Yaskawa INFORM job: R1_W17,20,22(0,0)OK-KM.JBI

/JOB
//NAME R1_W17,20,22(0,0)OK-KM
///FOLDERNAME KRIS-SCIANA
//POS
///NPOS 121,121,0,7,0,0
///TOOL 0
///POSTYPE PULSE
///PULSE
C00000=-189615,-139320,-99333,22908,80634,5417
C00001=-195814,-97363,-54861,18109,45254,4013
C00002=-195342,-89844,-49219,17779,45528,4291
C00003=-194630,-83582,-43444,17553,45059,4532
C00004=-193782,-82947,-43197,17110,45053,4932
C00005=-194630,-83582,-43444,17553,45059,4532
C00006=-194630,-82704,-41910,17701,44589,4439
C00007=-199143,-72536,-44097,19526,61527,3376
C00008=-199513,-75125,-46608,19573,61817,3281
C00009=-200501,-81674,-52788,19719,62464,3007
C00010=-207304,-71791,-24407,35263,30060,5319
C00011=-207149,-64591,-18647,35001,30129,5478
C00012=-204869,-60384,-14661,33643,29035,6515
C00013=-203452,-59589,-14281,32383,28672,7366
C00014=-204869,-60384,-14661,33643,29035,6515
C00015=-204869,-59185,-12583,34316,28482,6172
C00016=-204869,-60384,-14661,33643,29035,6515
C00017=-215068,-50959,-15594,37598,47140,3454
C00018=-215285,-50166,-15160,37584,47344,3432
C00019=-214356,-52683,-17577,37193,47111,3828
C00020=-214795,-55416,-20188,37217,47456,3749
C00021=-215972,-62244,-26544,37355,48272,3487
C00022=-217673,2073,-2688,-67811,68721,47040
C00023=-218977,3637,818,-67445,65858,48607
C00024=-219089,4523,1579,-67431,65778,48594
C00025=-218977,3637,818,-67445,65858,48607
C00026=-216731,7597,16575,-81534,66129,55483
C00027=-216731,8242,18363,-81863,65994,55863
C00028=-217587,5856,11870,-80689,65886,54435
C00029=-224554,-2275,-18337,-52519,68642,41010
C00030=-225245,-2625,-18625,-52307,68252,40859
C00031=-224554,-2275,-18337,-52519,68642,41010
C00032=-223707,-4148,-20438,-52681,69325,41069
C00033=-222614,-33118,-39506,-62827,46949,50873
C00034=-225738,-29129,-36820,-61092,45172,49948
C00035=-227041,-26413,-34946,-60254,44485,49501
C00036=-227207,-24592,-33670,-60039,44458,49378
C00037=-226942,-27472,-35680,-60383,44499,49577
C00038=-228936,-27670,-24586,-81470,38078,57242
C00039=-229553,-27860,-24718,-81378,37631,57193
C00040=-228393,-29098,-27492,-80247,38667,56535
C00041=-227197,-30656,-28257,-80893,39459,56892
C00042=-224091,-34376,-30000,-82400,41545,57754
C00043=-172648,-102914,-69268,-89134,45979,57650
C00044=-78280,-132294,-70134,-65050,82728,51954
C00045=231366,-50529,-85532,-14348,118547,17853
C00046=231331,-51716,-35505,-12276,87907,21200
C00047=229315,-48570,-29966,-12403,85849,20709
C00048=227923,-45606,-26730,-12487,85179,20296
C00049=227923,-45208,-25708,-12491,84764,20337
C00050=228522,-47247,-27691,-12456,85024,20518
C00051=199703,-85274,-38967,20911,45379,18978
C00052=198515,-84591,-38717,21283,45850,18535
C00053=199928,-86071,-39510,20852,45254,19054
C00054=200123,-88829,-42015,20735,45324,19162
C00055=200648,-95812,-48167,20467,45386,19423
C00056=223036,-16803,-12767,15055,51086,10558
C00057=223001,-10097,-5312,15317,49989,10370
C00058=221760,-6374,-575,16251,49262,9685
C00059=221760,-6023,569,16378,48758,9599
C00060=222987,-7382,-2234,15435,49509,10287
C00061=229840,2245,989,-2824,59416,19535
C00062=229297,2441,1158,-2588,59396,19324
C00063=229875,1901,-451,-2819,60125,19531
C00064=227161,1886,-1137,2630,57624,16683
C00065=227281,3372,123,2575,57604,16729
C00066=227129,1132,-3217,2621,58516,16692
C00067=227372,-1279,-6275,2488,59150,16802
C00068=228006,-7193,-13686,2154,60653,17078
C00069=231366,-50529,-85532,-14348,118547,17853
C00070=-77958,-132702,-65854,-64701,82399,51968
C00071=-138956,-107357,-30738,-74002,40113,39794
C00072=-140081,-59966,15635,-79359,38411,42592
C00073=-208206,-45897,20537,87676,15751,-45063
C00074=-207960,-49182,17085,86162,15646,-44311
C00075=-111965,-46340,36967,-74147,51082,48825
C00076=-82556,-17668,73730,-64807,60582,55576
C00077=-75120,-43857,42150,-58556,66417,53756
C00078=-148664,-83770,1112,-87446,33384,44594
C00079=-176147,-61139,7237,-80789,19096,34535
C00080=-180433,-47939,16447,-77543,16865,32116
C00081=-208028,-46200,20021,87142,15660,-44778
C00082=-207778,-49477,16583,85630,15556,-44027
C00083=-140712,-22447,70317,-98622,37333,53286
C00084=-126468,-40765,51508,-87063,43300,51710
C00085=-78280,-117024,-65873,-65050,51337,51954
C00086=204216,-84591,-49290,-51682,73827,23894
C00087=234941,-57799,-26790,-47858,90257,30629
C00088=199972,-101228,-53558,-4187,23841,10008
C00089=189033,-76626,-31890,10620,23559,1426
C00090=189033,-76626,-31890,10620,23559,1426
C00091=188864,-64798,-20049,11393,22392,1030
C00092=229125,-13360,-10863,-46798,76248,11937
C00093=228748,-14451,-12356,-46697,76301,11724
C00094=158433,-60990,9751,67845,21798,-31218
C00095=158927,-83907,-11161,65252,21999,-29865
C00096=192853,-97920,-56876,4665,27613,4814
C00097=204487,-80585,-57206,-6895,36944,11799
C00098=205889,-64287,-49388,-7540,40605,12218
C00099=203918,-48473,-33642,-6113,38883,11330
C00100=229115,-13382,-10880,-46798,76242,11935
C00101=228739,-14472,-12373,-46696,76295,11722
C00102=188637,-64887,-20002,11738,22348,831
C00103=195288,-76653,-33683,2057,24178,6381
C00104=224712,-65391,-70566,-27443,33176,35029
C00105=213770,-36542,-34460,77474,7084,-9175
C00106=213911,-28559,-27626,78111,6960,-9462
C00107=226738,-22872,-44138,-26151,38823,34122
C00108=225474,-24610,-45368,-24938,38325,33575
C00109=213819,-17629,4736,154767,14347,-43948
C00110=214272,-23134,1814,157793,15117,-45305
C00111=214272,-33613,-26176,108147,6753,-22913
C00112=214465,-33157,-25875,108062,6602,-22875
C00113=214484,-33168,-25884,108106,6590,-22894
C00114=214462,-14862,18245,165247,20516,-48770
C00115=217554,-35080,-3939,169426,16769,-50400
C00116=215729,-48765,-65733,21008,15669,16203
C00117=214456,-35235,-57699,21691,17865,16014
C00118=214365,-32785,-25079,110368,6760,-23908
C00119=218232,-57197,-39676,150711,6696,-41886
C00120=106022,-135537,-66235,115408,55550,-32403
BC00000=365100,2604,568777
BC00001=396813,15,501820
BC00002=396813,15,501820
BC00003=396813,15,501820
BC00004=396813,15,501820
BC00005=396813,15,501820
BC00006=396813,15,501820
BC00007=396813,15,501820
BC00008=396813,15,501820
BC00009=396813,15,501820
BC00010=289343,15,994506
BC00011=289343,15,994506
BC00012=289344,16,994504
BC00013=289344,16,994504
BC00014=289344,16,994504
BC00015=289344,16,994504
BC00016=289344,16,994504
BC00017=289343,15,994506
BC00018=289343,15,994506
BC00019=289343,15,994506
BC00020=289343,15,994506
BC00021=289343,15,994506
BC00022=398117,15,691553
BC00023=398117,15,691553
BC00024=398117,15,691553
BC00025=398117,15,691553
BC00026=398117,15,691553
BC00027=398117,15,691553
BC00028=398117,15,691553
BC00029=398117,15,691553
BC00030=398117,15,691553
BC00031=398117,15,691553
BC00032=398117,15,691553
BC00033=398174,15,1075175
BC00034=398174,15,1075175
BC00035=398174,15,1075175
BC00036=398174,15,1075175
BC00037=398174,15,1075175
BC00038=398174,15,1075175
BC00039=398174,15,1075175
BC00040=398174,15,1075175
BC00041=398174,15,1075175
BC00042=398174,15,1075175
BC00043=398174,15,1075175
BC00044=398174,15,1075175
BC00045=398174,29742,582568
BC00046=398174,29742,582568
BC00047=398174,29742,582568
BC00048=398174,29742,582568
BC00049=398174,29742,582568
BC00050=398174,29742,582568
BC00051=398174,29742,582568
BC00052=398174,29742,582568
BC00053=398174,29742,582568
BC00054=398174,29742,582568
BC00055=398174,29742,582568
BC00056=398174,24813,868263
BC00057=398174,24813,868263
BC00058=398174,24813,868263
BC00059=398174,24813,868263
BC00060=398174,24813,868263
BC00061=398174,24813,868263
BC00062=398174,24813,868263
BC00063=398174,24813,868263
BC00064=398174,24813,868263
BC00065=398174,24813,868263
BC00066=398174,24813,868263
BC00067=398174,24813,868263
BC00068=398174,24813,868263
BC00069=398174,29742,582568
BC00070=398174,15,1075175
BC00071=282653,15,945445
BC00072=282653,15,945445
BC00073=320510,15,961588
BC00074=320510,15,961588
BC00075=282653,15,931025
BC00076=282653,15,914571
BC00077=282653,15,945445
BC00078=282653,15,1075175
BC00079=282653,15,1075175
BC00080=282654,15,1075174
BC00081=282653,15,1075175
BC00082=282653,15,1075175
BC00083=282653,15,1075175
BC00084=282653,15,1075175
BC00085=398174,15,1075175
BC00086=344180,85519,956119
BC00087=344180,85519,956119
BC00088=331941,89333,813920
BC00089=331941,89333,813920
BC00090=331941,89333,813920
BC00091=331941,89333,813920
BC00092=363883,89134,716717
BC00093=363883,89134,716717
BC00094=331941,89333,813920
BC00095=331941,89333,813920
BC00096=331941,89333,813920
BC00097=331941,89333,813920
BC00098=331941,89333,813920
BC00099=331941,89333,813920
BC00100=331941,89333,813920
BC00101=331941,89333,813920
BC00102=331941,89333,813920
BC00103=331941,89333,813920
BC00104=398174,68400,1075175
BC00105=398174,60897,1075175
BC00106=398174,60897,1075175
BC00107=398174,60897,1075175
BC00108=398174,60897,1075175
BC00109=398174,60897,1075175
BC00110=398174,60897,1075175
BC00111=398174,60897,775711
BC00112=392644,57641,759002
BC00113=392644,57641,759002
BC00114=392644,57641,759002
BC00115=392644,57641,759002
BC00116=392644,57641,759002
BC00117=392644,57641,759002
BC00118=392644,57641,759002
BC00119=392644,57641,759002
BC00120=392644,373033,759002
///POSTYPE BASE
///RECTAN
///RCONF 0,0,0,0,1,0,0,0,0,0,0,0,0,0,0,0,0,0,0,0,0,0,0,0
P00006=2.006,1.622,-0.565,0.0000,0.0000,0.0000
P00021=0.073,2.058,-0.109,0.0000,0.0000,0.0000
P00022=2.006,1.622,-0.565,0.0000,0.0000,0.0000
///RCONF 0,0,0,0,0,0,0,0,0,0,0,0,0,0,0,0,0,0,0,0,0,0,0,0
P00023=-2.957,-4.083,2.762,0.0000,0.0000,0.0000
P00024=-1.466,-0.226,-0.419,0.0000,0.0000,0.0000
P00025=3.643,0.007,-2.585,0.0000,0.0000,0.0000
P00026=2.644,0.055,-2.583,0.0000,0.0000,0.0000
//INST
///DATE 2023/12/13 20:11
///ATTR SC,RW
///GROUP1 RB1,BS1
NOP
'r1_W17,20,22(0,0)
'Path S809 (for W415)
SFTOF
MOVJ C00000 BC00000 VJ=100.00
MOVJ C00001 BC00001 VJ=100.00
MOVJ C00002 BC00002 VJ=100.00
MOVL C00003 BC00003 V=60.0
REFP 3 C00004 BC00004
CALL JOB:SEARCH-R1
SET P021 P006
SFTON P021
MOVL C00005 BC00005 V=60.0
REFP 3 C00006 BC00006
CALL JOB:SEARCH-R1
SET P021 P006
SFTON P021
MOVL C00007 BC00007 V=60.0
MOVL C00008 BC00008 V=166.7
MOVL C00009 BC00009 V=166.7
'Path S811 (for W416)
SFTOF
MOVL C00010 BC00010 V=333.3
MOVJ C00011 BC00011 VJ=100.00
MOVL C00012 BC00012 V=60.0
REFP 3 C00013 BC00013
CALL JOB:SEARCH-R1
SET P022 P006
SFTON P022
MOVL C00014 BC00014 V=60.0
REFP 3 C00015 BC00015
CALL JOB:SEARCH-R1
SET P022 P006
SFTON P022
MOVL C00016 BC00016 V=60.0
MOVL C00017 BC00017 V=60.0
REFP 3 C00018 BC00018
CALL JOB:SEARCH-R1
SET P022 P006
SFTON P022
MOVL C00019 BC00019 V=60.0
MOVL C00020 BC00020 V=166.7
MOVL C00021 BC00021 V=166.7
'Path S814 (for W423)
SFTOF
MOVL C00022 BC00022 V=333.3
MOVL C00023 BC00023 V=60.0
REFP 3 C00024 BC00024
CALL JOB:SEARCH-R1
SET P025 P006
SFTON P025
MOVL C00025 BC00025 V=60.0
MOVL C00026 BC00026 V=60.0
REFP 3 C00027 BC00027
CALL JOB:SEARCH-R1
SET P025 P006
SFTON P025
MOVL C00028 BC00028 V=60.0
MOVL C00029 BC00029 V=60.0
REFP 3 C00030 BC00030
CALL JOB:SEARCH-R1
SET P025 P006
SFTON P025
MOVL C00031 BC00031 V=60.0
MOVL C00032 BC00032 V=166.7
'Path S815 (for W423)
SFTOF
MOVL C00033 BC00033 V=333.3
MOVL C00034 BC00034 V=166.7
MOVL C00035 BC00035 V=60.0
REFP 3 C00036 BC00036
CALL JOB:SEARCH-R1
SET P026 P006
SFTON P026
MOVL C00037 BC00037 V=60.0
MOVL C00038 BC00038 V=60.0
REFP 3 C00039 BC00039
CALL JOB:SEARCH-R1
SET P026 P006
SFTON P026
MOVL C00040 BC00040 V=60.0
MOVL C00041 BC00041 V=166.7
MOVL C00042 BC00042 V=166.7
MOVJ C00043 BC00043 VJ=100.00
'obrot 180
'Path VIA1089
SFTOF
MOVJ C00044 BC00044 VJ=100.00
'Path VIA1092
SFTOF
MOVJ C00045 BC00045 VJ=100.00
'Path S1093 (for W18)
SFTOF
MOVJ C00046 BC00046 VJ=100.00
MOVJ C00047 BC00047 VJ=100.00
MOVL C00048 BC00048 V=60.0
REFP 3 C00049 BC00049
CALL JOB:SEARCH-R1
SET P023 P006
SFTON P023
MOVL C00050 BC00050 V=60.0
MOVL C00051 BC00051 V=60.0
REFP 3 C00052 BC00052
CALL JOB:SEARCH-R1
SET P023 P006
SFTON P023
MOVL C00053 BC00053 V=60.0
MOVL C00054 BC00054 V=166.7
MOVL C00055 BC00055 V=166.7
'Path S1094 (for W18)
SFTOF
MOVJ C00056 BC00056 VJ=100.00
MOVJ C00057 BC00057 VJ=100.00
MOVL C00058 BC00058 V=60.0
REFP 3 C00059 BC00059
CALL JOB:SEARCH-R1
SET P024 P006
SFTON P024
MOVL C00060 BC00060 V=60.0
MOVL C00061 BC00061 V=60.0
REFP 3 C00062 BC00062
CALL JOB:SEARCH-R1
SET P024 P006
SFTON P024
MOVL C00063 BC00063 V=60.0
MOVL C00064 BC00064 V=60.0
REFP 3 C00065 BC00065
CALL JOB:SEARCH-R1
SET P024 P006
SFTON P024
MOVL C00066 BC00066 V=60.0
MOVL C00067 BC00067 V=166.7
MOVL C00068 BC00068 V=166.7
'Path VIA1095
SFTOF
MOVJ C00069 BC00069 VJ=100.00
'Path VIA1096
SFTOF
MOVJ C00070 BC00070 VJ=100.00
SFTON P022
MOVJ C00071 BC00071 VJ=100.00
MOVL C00072 BC00072 V=333.3 PL=0
REFP 1 C00073 BC00073
REFP 2 C00074 BC00074
MACRO1 MJ#(0) ARGF10
ARCON
MOVL C00075 BC00075 V=13.3
SFTON P021
MOVL C00076 BC00076 V=13.3
ARCOF
MOVL C00077 BC00077 V=250.0
SFTOF
'Path W415
SFTOF
SFTON P022
MOVJ C00078 BC00078 VJ=100.00
MOVJ C00079 BC00079 VJ=100.00
MOVL C00080 BC00080 V=100.0 PL=0
REFP 1 C00081 BC00081
REFP 2 C00082 BC00082
MACRO1 MJ#(0) ARGF10
ARCON
SFTON P021
MOVL C00083 BC00083 V=13.3
ARCOF
MOVL C00084 BC00084 V=166.7
SFTOF
'Path W1132
SFTOF
'Path VIA1097
SFTOF
MOVJ C00085 BC00085 VJ=100.00
'Path VIA1133
SFTOF
MOVJ C00086 BC00086 VJ=100.00
MOVJ C00087 BC00087 VJ=100.00
'Path W1098
SFTOF
'Path W1134
SFTOF
SFTON P023
MOVJ C00088 BC00088 VJ=100.00
MOVJ C00089 BC00089 VJ=100.00
MOVJ C00090 BC00090 VJ=100.00
MOVL C00091 BC00091 V=100.0 PL=0
REFP 1 C00092 BC00092
REFP 2 C00093 BC00093
MACRO1 MJ#(0) ARGF10
ARCON
SFTON P023
MOVL C00094 BC00094 V=13.3
ARCOF
TIMER T=0.50
MOVL C00095 BC00095 V=166.7
SFTOF
MOVJ C00096 BC00096 VJ=100.00
SFTON P024
MOVJ C00097 BC00097 VJ=100.00
MOVJ C00098 BC00098 VJ=100.00
MOVL C00099 BC00099 V=100.0 PL=0
REFP 1 C00100 BC00100
REFP 2 C00101 BC00101
MACRO1 MJ#(0) ARGF10
ARCON
SFTON P023
MOVL C00102 BC00102 V=13.3
ARCOF
MOVL C00103 BC00103 V=400.0
SFTOF
'Path W423
SFTOF
SFTON P026
MOVL C00104 BC00104 V=333.3
MOVL C00105 BC00105 V=166.7
MOVL C00106 BC00106 V=100.0 PL=0
REFP 1 C00107 BC00107
REFP 2 C00108 BC00108
MACRO1 MJ#(0) ARGF6
ARCON
MOVL C00109 BC00109 V=12.5
ARCOF
MOVL C00110 BC00110 V=166.7
SFTOF
MOVJ C00111 BC00111 VJ=100.00
SFTON P026
MOVJ C00112 BC00112 VJ=100.00
MACRO1 MJ#(0) ARGF6
MOVL C00113 BC00113 V=50.0 PL=0
ARCON
MOVL C00114 BC00114 V=12.5
ARCOF
TIMER T=1.00
SFTOF
MOVJ C00115 BC00115 VJ=100.00
MOVJ C00116 BC00116 VJ=25.00
SFTON P026
MOVJ C00117 BC00117 VJ=100.00
ARCON
MOVL C00118 BC00118 V=12.5
ARCOF
TIMER T=1.00
SFTOF
MOVL C00119 BC00119 V=166.7
SFTOF
MOVJ C00120 BC00120 VJ=100.00
END
